FUNCTION_BLOCK FB_MotionInterlocks IMPLEMENTS I_MotionInterlocks
VAR_INPUT
END_VAR
VAR_OUTPUT
END_VAR
VAR
    MotionSyncPrivateRef : REFERENCE TO FB_MotionSyncPrivate;
    (* Hardware *)
   // NC Forward Limit Switch: TRUE if ok to move
    bLimitForwardEnable AT %I*: BOOL;
    // NC Backward Limit Switch: TRUE if ok to move
    bLimitBackwardEnable AT %I*: BOOL;
    // NO Home Switch: TRUE if at home
    bHome AT %I*: BOOL;
   (* Psuedo-hardware *)
    // Forward enable EPS summary
    bAllForwardEnable: BOOL:=FALSE;
    // Backward enable EPS summary
    bAllBackwardEnable: BOOL:=FALSE;
    // Enable EPS summary encapsulating emergency stop button and any additional motion preventive hardware
    bAllEnable: BOOL:=FALSE;
    // Forward virtual gantry limit switch
    bGantryForwardEnable: BOOL:=FALSE;
    // Backward virtual gantry limit switch
    bGantryBackwardEnable: BOOL:=FALSE;
    // Set true to activate gantry EPS
    bGantryAxis: BOOL:=FALSE;
   // If TRUE, we want to enable the motor independently of PMPS or other safety systems.
    bPowerSelf: BOOL:=FALSE;
    // Determines when we automatically enable the motor
    nEnableMode: E_StageEnableMode:=E_StageEnableMode.DURING_MOTION;
    // Determines our encoder homing strategy
    nHomingMode: E_EpicsHomeCmd:=E_EpicsHomeCmd.NONE;
    // TRUE if we have safety permission to move
    bSafetyReady: BOOL;
    // TRUE if done enabling
    bEnableDone: BOOL;

   // NC STO Input: TRUE if ok to move
    {attribute 'pytmc' := '
        pv: PLC:bHardwareEnable
        io: i
        field: ZNAM FALSE
        field: ONAM TRUE
        field: DESC TRUE if STO not hit
    '}
    bHardwareEnable AT %I*: BOOL ;

    // Forward Enable EPS struct
    {attribute 'pytmc' := '
        pv: PLC:stEPSF
        io: i
        field: DESC Forward Enable Interlocks
    '}
    stEPSForwardEnable: DUT_EPS;
    // Backward Enable EPS struct
    {attribute 'pytmc' := '
        pv: PLC:stEPSB
        io: i
        field: DESC Backward Enable Interlocks
    '}
    stEPSBackwardEnable: DUT_EPS;
    // Power Enable EPS struct
    {attribute 'pytmc' := '
        pv: PLC:stEPSP
        io: i
        field: DESC Power Interlocks
    '}
    stEPSPowerEnable: DUT_EPS;

    // Used by the IOC to disable an axis
    {attribute 'pytmc' := '
        pv: PLC:bUserEnable
        io: io
        field: ZNAM DISABLE
        field: ONAM ENABLE
        field: DESC Used to disable power entirely for an axis
    '}
    bUserEnable: BOOL := TRUE;

    bLimOverride : BOOL;
    bSoftInterlock : BOOL;

    {attribute 'hide'}
    iMotionLogger 		: I_MotionLogger;

    {attribute 'hide'}
    bLocalExec : BOOL;
    {attribute 'hide'}
    bAllForwardEnabled: BOOL:=FALSE;
     {attribute 'hide'}
    bAllBackwardEnabled: BOOL:=FALSE;
    {attribute 'hide'}
    bAllEnabled: BOOL:=FALSE;
    {attribute 'hide'}
    bHomeBusy : BOOL;
    {attribute 'hide'}
    bMoveBusy	: BOOL;
    {attribute 'hide'}
    bNewMoveReq	: BOOL;
    {attribute 'hide'}
    bEnable: BOOL;
    {attribute 'hide'}
    bPrepareDisable : BOOL;

    {attribute 'hide'}
    bExecute : BOOL;
    {attribute 'hide'}
    bEPSOk : BOOL;

    {attribute 'hide'}
    sWarningMsg : STRING;
    {attribute 'hide'}
    nErpicsWarnId : UINT;
    {attribute 'hide'}
    bError : BOOL;
    {attribute 'hide'}
    bReset : BOOL;
    {attribute 'hide'}
    bLimHit : BOOL;
    {attribute 'hide'}
    bMoveDone : BOOL;
    {attribute 'hide'}
    eAxisState	: MC_AxisStates;
    {attribute 'hide'}
    ftForwardEnabled : F_TRIG;
    {attribute 'hide'}
    ftBackwardEnabled : F_TRIG;
    {attribute 'hide'}
    rtEnableMode : R_TRIG;
    {attribute 'hide'}
    rtStopExec : R_TRIG;
    {attribute 'hide'}
    rtNewMoveReq : R_TRIG;
    // reset cmds if done, error or reset
        {attribute 'hide'}
    rtDone : R_TRIG;
    {attribute 'hide'}
    rtError: R_TRIG;
    {attribute 'hide'}
    rtReset: R_TRIG;
    testVarRef : REFERENCE TO UINT;
END_VAR

// Read external private data
IF __ISVALIDREF(MotionSyncPrivateRef) THEN
    eAxisState := MotionSyncPrivateRef.SynPrvAxisState;
    bReset := MotionSyncPrivateRef.SynPrvReset;
    bError := MotionSyncPrivateRef.SynPrvError;
    bExecute := MotionSyncPrivateRef.SynPrvExec;
    bError := MotionSyncPrivateRef.SynPrvError;
    bHomeBusy := MotionSyncPrivateRef.SynPrvHomeBusy;
    bLocalExec := MotionSyncPrivateRef.SynPrvLocalExec;
    bMoveBusy := MotionSyncPrivateRef.SynPrvMoveBusy;
    bMoveDone := MotionSyncPrivateRef.SynPrvMoveDone;
    bNewMoveReq := MotionSyncPrivateRef.SynPrvNewMoveReq;
END_IF

bAllBackwardEnabled := bLimitBackwardEnable AND (bGantryBackwardEnable OR NOT bGantryAxis) AND stEPSForwardEnable.bEPS_OK;
bAllForwardEnabled := bLimitForwardEnable AND (bGantryForwardEnable OR NOT bGantryAxis) AND stEPSBackwardEnable.bEPS_OK;
/////////////////////////////////////////////////////////////////////////////
// SoftInterlock is a user defined interloc logic active high
/////////////////////////////////////////////////////////////////////////////
bAllEnabled := bEnable AND bHardwareEnable AND stEPSPowerEnable.bEPS_OK AND NOT bSoftInterlock;
bAllEnabled R= NOT bUserEnable OR bSoftInterlock;
//// use falling trigger to avoid spaming  sErrorMessage
ftForwardEnabled(CLK:=bAllForwardEnabled);
ftBackwardEnabled(CLK:=bAllBackwardEnabled);
///////////////////////////////////////////////////////////////
// Raise a warning when limit are hit outisde of homing routine
///////////////////////////////////////////////////////////////
IF   ftForwardEnabled.Q OR ftBackwardEnabled.Q THEN
    // Not an error, just a warning
    IF NOT bAllForwardEnabled THEN
        sWarningMsg:='Cannot move past positive limit.';
    ELSIF NOT bAllBackwardEnabled THEN
        sWarningMsg:='Cannot move past Negative limit.';
    END_IF
    bLimHit := TRUE;
    // will serve later
    bLimOverride := TRUE;
END_IF

bPrepareDisable R= bNewMoveReq;
// Moves are automatically allowed if no safety hooks. Otherwise, some other code will set this.
bSafetyReady S= bPowerSelf;

rtNewMoveReq(CLK:=bNewMoveReq);
rtEnableMode(CLK:=(EnableMode = E_StageEnableMode.DURING_MOTION));
// Handle auto-enable timing
CASE EnableMode OF
    E_StageEnableMode.ALWAYS:
        bEnable:=TRUE;
    E_StageEnableMode.DURING_MOTION:
        IF rtEnableMode.Q THEN
            bEnable := FALSE;
        END_IF
        // Power interlock only enabled with a new move request
        IF rtNewMoveReq.Q THEN
            bEnable S= bSafetyReady;
        END_IF
END_CASE

// Get a definitive bEnabled reading
CASE eAxisState OF
    // We are not enabled if there is an issue
    MC_AXISSTATE_UNDEFINED, MC_AXISSTATE_DISABLED, MC_AXISSTATE_ERRORSTOP:
        bEnableDone := FALSE;
    ELSE
        bEnableDone := TRUE;
END_CASE

// This is the output interlock check used to allow the requested move
bLocalExec:= bExecute AND bAllEnabled AND bEnableDone AND bSafetyReady;

// when move is done, interupted or target reached disabled drive after axis has settle
rtStopExec(CLK:=bMoveDone);
// Handle auto-disable timing
bPrepareDisable S= (EnableMode = E_StageEnableMode.DURING_MOTION ) AND rtStopExec.Q;
// Delay the disable until we reach standstill, else brake issues or other race conditions
IF bPrepareDisable AND ( eAxisState = MC_AXISSTATE_STANDSTILL ) THEN
    bPrepareDisable := FALSE;
    bEnable := FALSE;
END_IF

// Prepare next move
bMoveDone := FALSE;

// react to reset if the axis is standstill ( clearing error )
IF bReset THEN
    bLimOverride := FALSE;
    bLimHit := FALSE;
    bReset := FALSE;
    bError := FALSE;
END_IF

IF bError THEN
    bEnable := FALSE;
END_IF

// write external private data
IF __ISVALIDREF(MotionSyncPrivateRef) THEN
    // control power based on interlocks
    MotionSyncPrivateRef.SynPrvAllEn := bAllEnable;
    MotionSyncPrivateRef.SynPrvAllBwdEn := bAllBackwardEnable;
    MotionSyncPrivateRef.SynPrvAllFwdEn := bAllForwardEnable;
    MotionSyncPrivateRef.SynPrvLimBwd := bLimitForwardEnable;
    MotionSyncPrivateRef.SynPrvLimFwd := bLimitBackwardEnable;
    MotionSyncPrivateRef.SynPrvHome := bHome;
    MotionSyncPrivateRef.SynPrvLimHit := bLimHit;
END_IF

PROPERTY AllBackwardEnabled : BOOL
GET
AllBackwardEnabled  := bAllBackwardEnabled ;
END_GET
END_PROPERTY

PROPERTY AllEnabled : BOOL
GET
AllEnabled := bAllEnabled;
END_GET
END_PROPERTY

PROPERTY AllForwardEnabled : BOOL
GET
AllForwardEnabled  := bAllForwardEnabled ;
END_GET
END_PROPERTY

{attribute 'monitoring':= 'variable'}
PROPERTY EnableDone : BOOL
GET
END_GET
END_PROPERTY

{attribute 'monitoring':= 'variable'}
PROPERTY EnableMode : E_StageEnableMode
GET
EnableMode := nEnableMode;
END_GET
SET
nEnableMode := EnableMode;
END_SET
END_PROPERTY

PROPERTY EPSBackwardEnable : BOOL
GET
EPSBackwardEnable := stEPSBackwardEnable.bEPS_OK;
END_GET
SET
stEPSBackwardEnable.bEPS_OK := EPSBackwardEnable;
END_SET
END_PROPERTY

PROPERTY EPSForwardEnable : BOOL
GET
EPSForwardEnable := stEPSForwardEnable.bEPS_OK;
END_GET
SET
stEPSForwardEnable.bEPS_OK := EPSForwardEnable;
END_SET
END_PROPERTY

{attribute 'monitoring':= 'variable'}
PROPERTY EPSPowerEnable : BOOL
GET
EPSPowerEnable := stEPSPowerEnable.bEPS_OK;
END_GET
SET
stEPSPowerEnable.bEPS_OK := EPSPowerEnable;
END_SET
END_PROPERTY

//FB_Init is always available implicitly and it is used primarily for initialization.
//The return value is not evaluated. For a specific influence, you can also declare the
//methods explicitly and provide additional code there with the standard initialization
//code. You can evaluate the return value.
METHOD FB_Init: BOOL
VAR_INPUT
    bInitRetains: BOOL; // TRUE: the retain variables are initialized (reset warm / reset cold)
    bInCopyCode: BOOL;  // TRUE: the instance will be copied to the copy code afterward (online change)
    iMotionLogger 		: I_MotionLogger;
END_VAR
THIS^.iMotionLogger := iMotionLogger;
END_METHOD

PROPERTY GantryAxis : BOOL
GET
 GantryAxis :=  bGantryAxis;
END_GET
SET
 bGantryAxis :=  bGantryAxis;
END_SET
END_PROPERTY

PROPERTY GantryBackwardEnable : BOOL
GET
GantryBackwardEnable := bGantryBackwardEnable;
END_GET
SET
bGantryBackwardEnable := GantryBackwardEnable;
END_SET
END_PROPERTY

PROPERTY GantryForwardEnable : BOOL
GET
GantryForwardEnable := bGantryForwardEnable;
END_GET
SET
bGantryForwardEnable := GantryForwardEnable;
END_SET
END_PROPERTY

{attribute 'monitoring':= 'variable'}
PROPERTY HardwareEnable : BOOL
GET
HardwareEnable :=  bHardwareEnable;
END_GET
SET
bHardwareEnable := HardwareEnable;
END_SET
END_PROPERTY

PROPERTY LimBwdEnable : BOOL
GET
LimBwdEnable := bLimitBackwardEnable;
END_GET
SET
bLimitBackwardEnable := LimBwdEnable;
END_SET
END_PROPERTY

PROPERTY LimFwdEnable : BOOL
GET
LimFwdEnable := bLimitForwardEnable;
END_GET
SET
bLimitForwardEnable := LimFwdEnable;
END_SET
END_PROPERTY

{attribute 'monitoring':= 'variable'}
PROPERTY LimHit : BOOL
GET
LimHit := bLimHit;
END_GET
END_PROPERTY

PROPERTY LimHome : BOOL
GET
END_GET
SET
END_SET
END_PROPERTY

PROPERTY LimOverride : BOOL
GET
END_GET
END_PROPERTY

PROPERTY INTERNAL MotionSyncPrivate : REFERENCE TO FB_MotionSyncPrivate
GET
MotionSyncPrivate := MotionSyncPrivateRef;
END_GET
SET
MotionSyncPrivateRef REF= MotionSyncPrivate;
END_SET
END_PROPERTY

PROPERTY PowerSelf : BOOL
GET
 PowerSelf := bPowerSelf;
END_GET
SET
 bPowerSelf := PowerSelf;
END_SET
END_PROPERTY

{attribute 'monitoring':= 'variable'}
PROPERTY PrepareDisable : BOOL
GET
PrepareDisable := bPrepareDisable;
END_GET
END_PROPERTY

PROPERTY SafetyReady : BOOL
GET
SafetyReady := bSafetyReady;
END_GET
SET
bSafetyReady := SafetyReady;
END_SET
END_PROPERTY

PROPERTY SoftInterlock : BOOL
GET
SoftInterlock := bSoftInterlock;
END_GET
SET
bSoftInterlock := SoftInterlock;
END_SET
END_PROPERTY

PROPERTY INTERNAL TestStates : MC_AxisStates
GET
END_GET
SET
END_SET
END_PROPERTY

{attribute 'monitoring':= 'variable'}
PROPERTY UserEnable : BOOL
GET
UserEnable := bUserEnable;
END_GET
END_PROPERTY

PROPERTY WarnID : UINT
GET
WarnID  := nErpicsWarnId;
END_GET
END_PROPERTY

{attribute 'monitoring':= 'variable'}
PROPERTY WarningMsg : STRING
GET
WarningMsg := sWarningMsg;
END_GET
END_PROPERTY

END_FUNCTION_BLOCK

(* stored: Version 1.1.0.1
   POU FB_MotionInterlocks: Id {875748a6-e3b4-4780-a711-0e1eb4182bc0}, SpecialFunc None
   Property AllBackwardEnabled: Id {418fcf62-072d-4be6-9a52-23305e127201}
   Get Get: Id {55a054b8-413b-4eb9-bcde-040b97b12037}
   Property AllEnabled: Id {b8e0c844-5e14-430a-80f0-4b68fea05847}
   Get Get: Id {6ea43e2c-0382-4571-9cfc-7bb729ee79e3}
   Property AllForwardEnabled: Id {2f7747e3-44e7-42e0-9a1c-83d2d1a76054}
   Get Get: Id {1ca1d849-7776-4ef6-9a28-190e986cc112}
   Property EnableDone: Id {e8f686cf-2820-4def-9cf3-b4656f653df8}
   Get Get: Id {08422664-dee5-4efb-b45d-daa37c0a0460}
   Property EnableMode: Id {0059a3f0-809f-424e-ade1-142436c73b96}
   Get Get: Id {c252aba3-058d-4c88-b3ae-fd371338d57a}
   Set Set: Id {d7a5f3e4-7958-4366-80c3-d36a1f1d8bfd}
   Property EPSBackwardEnable: Id {946334c8-7a18-4f9f-949c-41f8e1008952}
   Get Get: Id {578cc864-6d35-4e4b-b60c-d4a4c932b7f7}
   Set Set: Id {86306b68-3cd4-4e6e-94fa-989b1a36f95a}
   Property EPSForwardEnable: Id {f4160bfd-86cc-47bf-8643-0b6329df5bb5}
   Get Get: Id {e7e6fb72-a940-4240-94e8-ba0f5b5f069a}
   Set Set: Id {e348ff27-726d-4eb3-8dd3-7358973ba387}
   Property EPSPowerEnable: Id {92783980-27d5-4db6-93ad-759db6eb8d88}
   Get Get: Id {5901b928-70bf-45c0-9664-fb5466a768f0}
   Set Set: Id {d5afccd0-d5e1-4ad6-8d85-c44d6f4e523c}
   Method FB_Init: Id {84019423-7ce0-4649-83b3-d87beaa3ba25}
   Property GantryAxis: Id {d8cb5e8d-9253-42f7-9db8-070eb5987299}
   Get Get: Id {90d116f0-2ada-46f1-bf3e-472f395eedca}
   Set Set: Id {1abb758b-9861-482a-a859-5ba04c1504b8}
   Property GantryBackwardEnable: Id {6eb9203e-9a27-4754-832f-3e6ac487d7cd}
   Get Get: Id {c16b98fb-bd19-41f8-8513-af8b053105c4}
   Set Set: Id {411048ad-2cbc-4674-9fb4-645d69a609a3}
   Property GantryForwardEnable: Id {49ac7373-d315-4647-997e-c3d4fbe89b3d}
   Get Get: Id {f431d19d-5fc7-4cdb-b93c-67ea289b1b4a}
   Set Set: Id {0282b8e9-d635-4cf4-8302-0e014dc947a3}
   Property HardwareEnable: Id {e3e787d4-24da-4bb1-8e05-fc15966309ef}
   Get Get: Id {89427268-48d1-4a1e-8c9b-5535b2e74a3b}
   Set Set: Id {1c449a44-7513-4afc-ad7e-ad4e152db2dd}
   Property LimBwdEnable: Id {f0c12a5c-c1fb-43de-bba5-3d0b5a489e5e}
   Get Get: Id {37912160-1a31-42d9-94e4-e0d17cedefed}
   Set Set: Id {cf37b50f-e07e-4d56-aee1-bdbbb25c2090}
   Property LimFwdEnable: Id {bad98783-f68c-4f18-8ede-2f4301263843}
   Get Get: Id {68c7fce3-79d3-4024-9097-1684f0f11d11}
   Set Set: Id {16df96f9-94f0-4d35-9b1c-fda03f8469e0}
   Property LimHit: Id {42c9b53e-e670-4408-8538-d34ff8b98535}
   Get Get: Id {a3588f8d-5778-455b-960b-1464f8c08488}
   Property LimHome: Id {98a7960f-d5b5-4afa-a6d4-836668115fc2}
   Get Get: Id {f1ca984e-77a2-439a-be50-7890b12815a4}
   Set Set: Id {390937c7-0fb9-46a6-a140-1f6dc26be67b}
   Property LimOverride: Id {acaf48e7-e68f-469d-af64-e985b96c68e0}
   Get Get: Id {46ed310e-8e71-479e-beb0-02beb59809d3}
   Property MotionSyncPrivate: Id {c5b0c731-4cdc-4ae0-99fc-43a250afbbac}
   Get Get: Id {be314522-61b0-498a-873d-558733e1fa67}
   Set Set: Id {e18cbaf1-1537-47a9-a31a-7ffa5ed29a91}
   Property PowerSelf: Id {fb36e9c1-0ee1-4f1a-b06f-22d945195377}
   Get Get: Id {c06ff4fd-ee59-4911-94a2-c723bdd82017}
   Set Set: Id {b9461afa-a4ea-4cd5-ab04-03c92360ffde}
   Property PrepareDisable: Id {74f72c04-fe7f-4e73-bd9e-9da711ed7881}
   Get Get: Id {fed14a6f-2527-439a-8476-ab4afab54f62}
   Property SafetyReady: Id {62e38fe3-a7fb-4294-903f-29b79adc8e09}
   Get Get: Id {827e9c82-e09d-4f11-ade7-bddb9139debf}
   Set Set: Id {f2385fd1-8c86-450d-ac93-4fa797c9b41c}
   Property SoftInterlock: Id {4ee885b6-25d1-4fb2-a46f-f025c9b60b25}
   Get Get: Id {eb06040e-af5f-494a-8ce8-85ea788d7e96}
   Set Set: Id {7b058ca7-724e-487e-af3c-51195cf468a3}
   Property TestStates: Id {aaf9585c-9ff4-4821-b470-d1b30fe7326a}
   Get Get: Id {32fdf0ba-3841-4831-94ee-d0715a7ed1be}
   Set Set: Id {92293fb7-21b5-47c3-a969-81bb0f21c9c1}
   Property UserEnable: Id {7e460973-7eca-4640-a87e-aea5109100a1}
   Get Get: Id {60a2a96e-359c-44c0-b656-b6511b040c6b}
   Property WarnID: Id {5598e3c0-c025-4591-a33e-0591f1851621}
   Get Get: Id {37a33505-3c15-43ab-b9e2-da7fe440eb0c}
   Property WarningMsg: Id {c58a222e-888c-449d-acb8-7036a45dc5e8}
   Get Get: Id {c813683b-22cc-422c-89ed-ba893df5d926} *)
